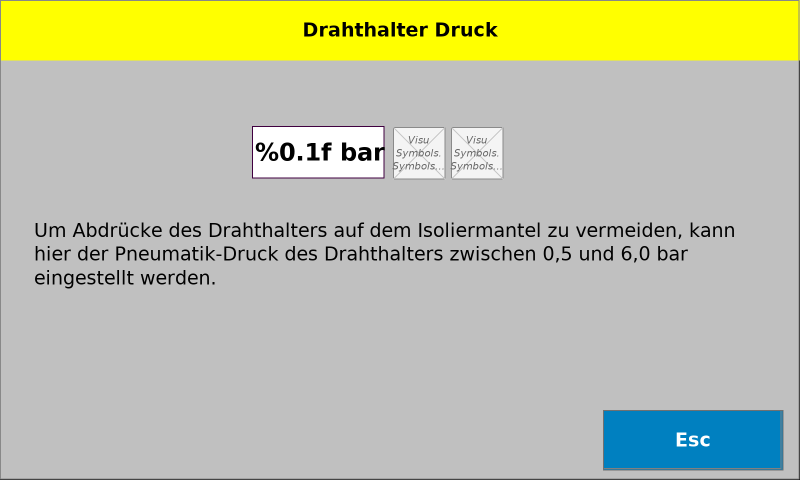
VISUALIZATION DrahthalterDruck  // 800x480
    Rectangle (0,0 800x480)
    Rectangle (0,0 800x60), "Drahthalter Druck"
    Button (603,410 180x60), "Esc"
        OnMouseUp: change screen: Previous 
    Rectangle (252,126 132x52), "%0.1f bar", text variable: DB6.rDrahthalterSchliessdruck
    Image (393,127 52x52), image: VisuSymbols.Symbols.TriangleLeft
        OnMouseClick: execute { P_DecDruck(); }
    Image (451,127 52x52), image: VisuSymbols.Symbols.TriangleRight
        OnMouseClick: execute { P_IncDruck(); }
    Label (31,192 730x124), "Um Abdrücke des Drahthalters auf dem Isoliermantel zu vermeiden, kann hier der Pneumatik-Druck des Drahthalters zwischen 0,5 und 6,0 bar eingestellt werden."
END_VISUALIZATION

(* stored: Version 1.1.0.1, ProductVersion 3.1.4024.3
   Visu DrahthalterDruck: Id {8d99618b-fa0c-4e8c-a9e0-35a6be34df82} *)
